(* PLC project Unnamed, Unknown Unnamed 1 *)
(* stored: creationDateTime 2025-04-20T22:58:20, modificationDateTime 2025-04-29T23:09:04 *)

TYPE matrix : ARRAY[0..3] OF DINT := [1, 2, 3, 4];
END_TYPE

FUNCTION_BLOCK element_selector
  VAR_INPUT
    M : matrix;
    index : UINT;
  END_VAR
  VAR_OUTPUT
    out : DINT;
  END_VAR

            out := M[index];

          
END_FUNCTION_BLOCK

FUNCTION_BLOCK element_setter
  VAR_IN_OUT
    M : matrix;
  END_VAR
  VAR_INPUT
    index : UINT;
    value : DINT;
  END_VAR
  VAR_OUTPUT
    out : DINT;
  END_VAR

            M[index] := value;
out := M[index];
          
END_FUNCTION_BLOCK

PROGRAM matrix_mul
  VAR
    m_A : matrix := [1, 2, 3, 4];
    m_B : matrix := [1, 2, 3, 4];
    m_C : matrix;
  END_VAR
  VAR
    i AT %QW0 : UINT := 0;
    j AT %QW1 : UINT := 0;
    k AT %QW2 : UINT := 0;
    n AT %QW3 : UINT := 2;
    index_A AT %QW4 : UINT;
    index_B AT %QW5 : UINT;
    index_C AT %QW6 : UINT;
    element_a AT %MD0 : DINT;
    element_b AT %MD1 : DINT;
    element_c AT %MD2 : DINT;
    check AT %MD3 : DINT;
    run_flag AT %IX0.0 : BOOL := true;
  END_VAR
  VAR
    input_matrices0 : element_selector;
    input_matrices1 : element_selector;
    element_setter0 : element_setter;
    element_selector0 : element_selector;
    element_selector1 : element_selector;
    element_selector2 : element_selector;
    element_selector3 : element_selector;
  END_VAR
  VAR  (* added by the conversion: wires and edge detectors of the diagram *)
    _GE48_ENO : BOOL;
    _GE48_OUT : BOOL;
    _MUL43_ENO : BOOL;
    _MUL43_OUT : UINT;
    _MUL6_ENO : BOOL;
    _MUL6_OUT : UINT;
    _MUL19_ENO : BOOL;
    _MUL19_OUT : UINT;
    _MOVE49_ENO : BOOL;
    _MOVE49_OUT : UINT;
    _GE34_ENO : BOOL;
    _GE34_OUT : BOOL;
    _MOVE40_ENO : BOOL;
    _MOVE40_OUT : UINT;
    _GE52_ENO : BOOL;
    _GE52_OUT : BOOL;
    _MUL68_ENO : BOOL;
    _MUL68_OUT : DINT;
  END_VAR

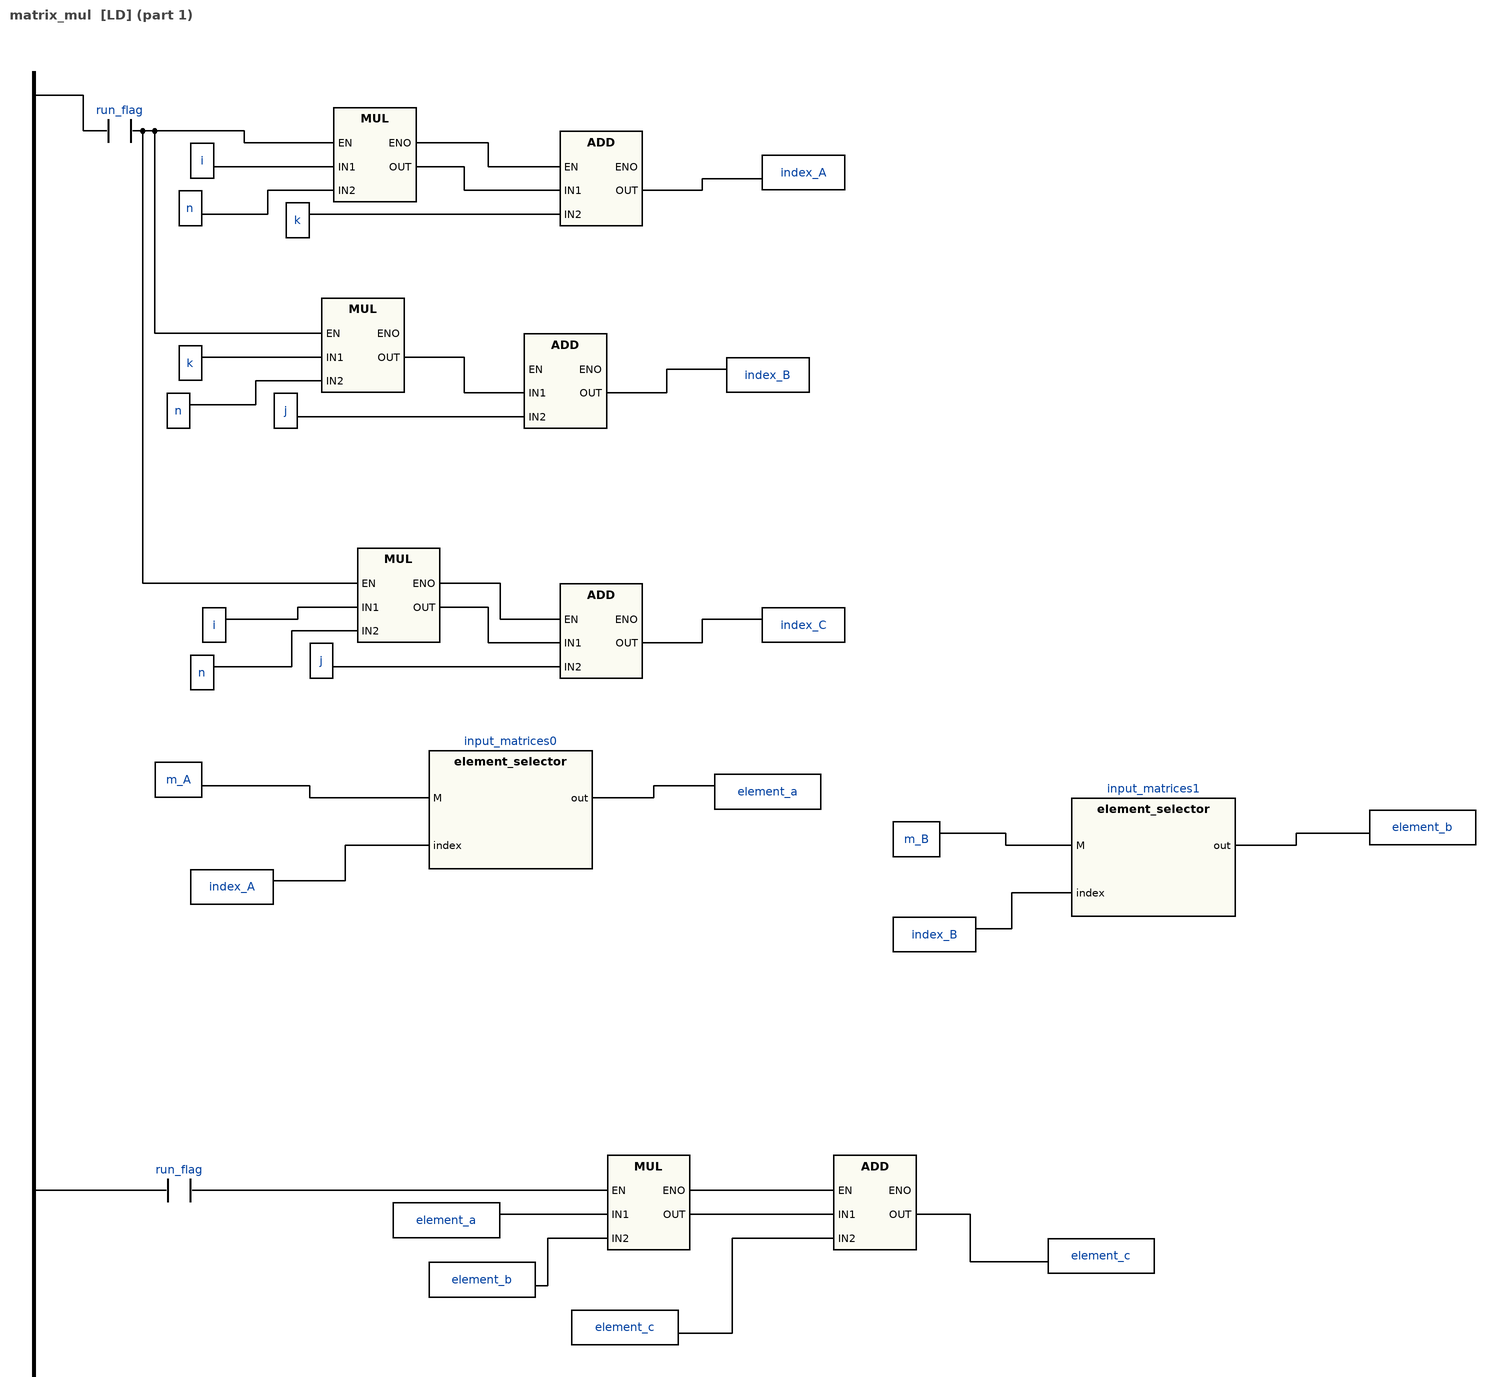
(* LD diagram, written out as Structured Text *)
input_matrices0(M := m_A, index := index_A);
element_a := input_matrices0.out;
input_matrices1(M := m_B, index := index_B);
element_b := input_matrices1.out;
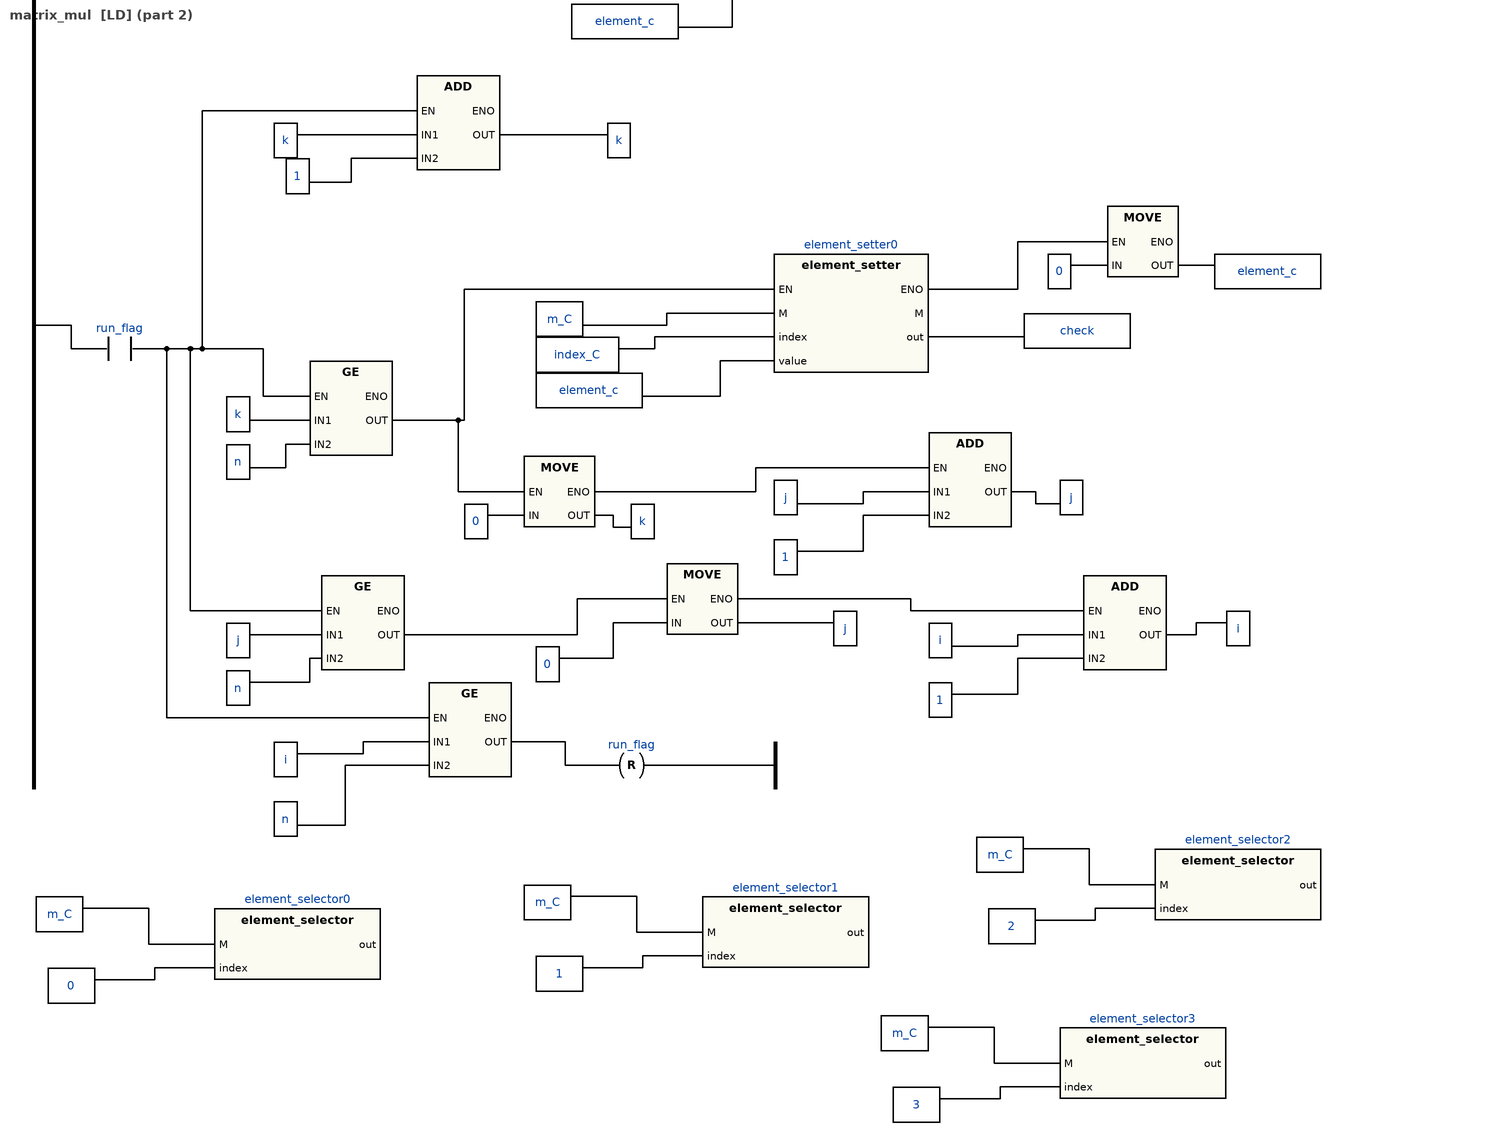
_GE48_OUT := GE(EN := run_flag, IN1 := k, IN2 := n, ENO => _GE48_ENO);
element_setter0(EN := _GE48_OUT, M := m_C, index := index_C, value := element_c);
IF element_setter0.ENO THEN check := element_setter0.out; END_IF;
_MUL43_OUT := MUL(EN := run_flag, IN1 := i, IN2 := n, ENO => _MUL43_ENO);
IF _MUL43_ENO THEN index_A := _MUL43_OUT + k; END_IF;
_MUL6_OUT := MUL(EN := run_flag, IN1 := k, IN2 := n, ENO => _MUL6_ENO);
index_B := _MUL6_OUT + j;
_MUL19_OUT := MUL(EN := run_flag, IN1 := i, IN2 := n, ENO => _MUL19_ENO);
IF _MUL19_ENO THEN index_C := _MUL19_OUT + j; END_IF;
IF run_flag THEN k := k + 1; END_IF;
_MOVE49_OUT := MOVE(EN := _GE48_OUT, IN := 0, ENO => _MOVE49_ENO);
IF _MOVE49_ENO THEN k := _MOVE49_OUT; END_IF;
IF _MOVE49_ENO THEN j := j + 1; END_IF;
_GE34_OUT := GE(EN := run_flag, IN1 := j, IN2 := n, ENO => _GE34_ENO);
_MOVE40_OUT := MOVE(EN := _GE34_OUT, IN := 0, ENO => _MOVE40_ENO);
IF _MOVE40_ENO THEN j := _MOVE40_OUT; END_IF;
IF _MOVE40_ENO THEN i := i + 1; END_IF;
_GE52_OUT := GE(EN := run_flag, IN1 := i, IN2 := n, ENO => _GE52_ENO);
IF _GE52_OUT THEN run_flag := FALSE; END_IF;
_MUL68_OUT := MUL(EN := run_flag, IN1 := element_a, IN2 := element_b, ENO => _MUL68_ENO);
IF _MUL68_ENO THEN element_c := _MUL68_OUT + element_c; END_IF;
IF element_setter0.ENO THEN element_c := 0; END_IF;
element_selector0(M := m_C, index := 0);
element_selector1(M := m_C, index := 1);
element_selector2(M := m_C, index := 2);
element_selector3(M := m_C, index := 3);
END_PROGRAM

CONFIGURATION Config0
  RESOURCE Res0 ON PLC
    TASK task0(INTERVAL := T#3s, PRIORITY := 0);
    PROGRAM instance0 WITH task0 : matrix_mul;
  END_RESOURCE
END_CONFIGURATION
